// TIA Portal V21 export
TYPE "Std_SezionePastorizzatore"
   STRUCT
      Spare : Bool;
   END_STRUCT;
END_TYPE
